SUBAPPLICATION Uebung_076 (* MSS mit Compound Scaling auf UT ausgeben *)
  (* Standard: 61499-2; Description: Copyright (c) 2023 Meisterschulen am Ostbahnhof This program and the accompanying materials are made available under the terms of the Eclipse Public License 2.0 which is available at https://www.eclipse.org/legal/epl-2.0/ SPDX-License-Identifier: EPL-2.0 *)
  (* Version 1.0, 2026-06-01, Franz Höpfinger, Meisterschulen am Ostbahnhof, MSS Machine Selected Speed mit Compound Scaling (0.256 upper / 0.001 lower) *)
  PACKAGE Uebungen;
  IMPORT Uebungen::const::UT::TECU::DefaultPool_TECU_Numeric::NumberVariable_Wheel_based_machine_speed_N;
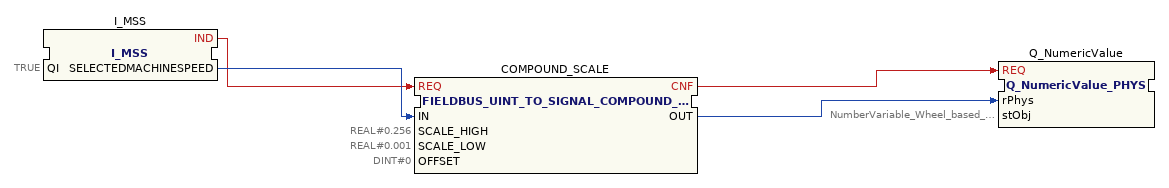
  (* TODO: NumberVariable_Machine_selected_speed im Object Pool anlegen, und hier umändern. solange verwenden wir hier NumberVariable_Wheel_based_machine_speed ersatzweise *)
  FBS
    I_MSS : isobus::tecu::I_MSS(QI := TRUE);
    COMPOUND_SCALE : logiBUS::signalprocessing::fieldbus::FIELDBUS_UINT_TO_SIGNAL_COMPOUND_SCALE(SCALE_HIGH := REAL#0.256, SCALE_LOW := REAL#0.001, OFFSET := DINT#0);
    Q_NumericValue : isobus::UT::Q::Q_NumericValue_PHYS(stObj := NumberVariable_Wheel_based_machine_speed_N);
  END_FBS
  EVENT_CONNECTIONS
    I_MSS.IND TO COMPOUND_SCALE.REQ;
    COMPOUND_SCALE.CNF TO Q_NumericValue.REQ;
  END_CONNECTIONS
  DATA_CONNECTIONS
    I_MSS.SELECTEDMACHINESPEED TO COMPOUND_SCALE.IN;
    COMPOUND_SCALE.OUT TO Q_NumericValue.rPhys;
  END_CONNECTIONS
END_SUBAPPLICATION
